{attribute 'GeneratedUsingTerminal: EPP3632-0001-0016'}
{attribute addProperty BoxType "EPP3632-0001-0016"}
{attribute addProperty Id "Ch2_ValueAT %I*INT2"}
{attribute addProperty CRC "2674427622"}
{attribute addProperty Size "2"}
TYPE Ch2_Sample_9F6886E6 EXTENDS InputBase_8311D824 :
STRUCT
	{attribute addProperty Name "Ch2_Value"}
	Ch2_Value AT %I* : INT;
END_STRUCT
END_TYPE

(* stored: Version 1.2.0.0, ProductVersion 3.1.4024.9
   DUT Ch2_Sample_9F6886E6: Id {2fec5754-873f-429c-a73b-e99d6f327208} *)
